FUNCTION_BLOCK PMLStateMachine IMPLEMENTS IPmlStateMachine
VAR_INPUT
END_VAR
VAR_OUTPUT
END_VAR
VAR
	_pmlStateMachine : Tc3_PackML_V2.PML_StateMachine;
	_pmlModeMachine : Tc3_PackML_V2.PML_UnitModeManager;
	_subUnits : ARRAY[0..9] OF IPmlStateMachine;
	_SubUnitReference: ST_PMLSubUnitInfoRef;
	i: DINT;
END_VAR


_pmlStateMachine(eMode := _pmlModeMachine.eModeStatus, stSubUnitInfoRef := _SubUnitReference);
_pmlModeMachine(eState := _pmlStateMachine.eState);

METHOD PUBLIC GetCurrentMode : E_PmlProtectedUnitMode
VAR_INPUT
END_VAR
GetCurrentMode := _pmlModeMachine.eModeStatus;
END_METHOD

METHOD PUBLIC GetCurrentState : E_PMLState
VAR_INPUT
END_VAR
GetCurrentState := _pmlStateMachine.eState;
END_METHOD

METHOD PUBLIC PmlModeCommand : Bool
VAR_INPUT
	Mode : E_PMLProtectedUnitMode;
END_VAR
_pmlModeMachine.eModeCommand := Mode;
END_METHOD

METHOD PUBLIC PmlStateCommand : BOOL
VAR_INPUT
	Command : E_PMLCommand;
END_VAR
_pmlStateMachine.eCommand := Command;
END_METHOD

METHOD PUBLIC RegisterSubUnit : IPmlStateMachine
VAR_INPUT
	SubUnit : IPmlStateMachine;
END_VAR
FOR i := 0 TO UPPER_BOUND(_subUnits,1) DO
	IF _subUnits[i] = 0 THEN
		_subUnits[i] := SubUnit;
	END_IF
END_FOR
END_METHOD

METHOD PUBLIC SetStateComplete : BOOL
VAR_INPUT
END_VAR
_pmlStateMachine.M_StateComplete();
END_METHOD

END_FUNCTION_BLOCK

(* stored: Version 1.1.0.1, ProductVersion 3.1.4024.12
   POU PMLStateMachine: Id {60400ea6-a6d0-4d71-8555-f15b7929c342}, SpecialFunc None
   Method GetCurrentMode: Id {a328d1d9-ecc8-4538-a2cc-179227c6ea57}
   Method GetCurrentState: Id {8c64c6da-7bfe-4eb7-ad2f-8614ebc2ae80}
   Method PmlModeCommand: Id {8f9efc6b-7148-4714-b677-c65effb81184}
   Method PmlStateCommand: Id {54af98e0-d3e9-44c6-81e2-5076efd7e22a}
   Method RegisterSubUnit: Id {2bdb4e5c-f6a3-4bbf-b17b-def1b8843c9f}
   Method SetStateComplete: Id {ca883fc1-f163-42f5-8b56-82749a1c7d47} *)
